{attribute 'Tc2GvlVarNames'}
{attribute 'strict'}
//Tipologia di Magazzino Falde
TYPE e_Tipo_Magazzino_Falde :
(
	NOT_DEFINED				:= -1,
	(* Magazzino Falde Per Pallettizzatore PACCHI*)
	//MAGAZZINO_FALDE_CENTRO_FISSO 		:= 1, //LA Y DI PRELIEVO RIMANE COSTANTE PER OGNI FORMATO
	//MAGAZZINO_FALDE_CENTRO_VARIABILE  	:= 2, //LA Y DI PRELIEVO SI ADATTA AL FORMATO DELLA FALDA
	
	(* Magazzino Falde per Pallettizzatore LASTRE*)
	MAGAZZINO_FALDE_IN_WA		 := 10, 	(* Identifica che il magazzino delle falde è una WorkArea *) 
	MAGAZZINO_FALDE_IN_PP		 := 20	 	(* Identifica che il magazzino delle falde è un Pick-Point, quindi elemento statico non asservito da LGV *) 

);
END_TYPE
//  NOT_DEFINED = '-1'

(* stored: Version 1.1.0.1, ProductVersion 3.1.4024.11
   EnumerationTextList e_Tipo_Magazzino_Falde: Id {26c1fc94-ade3-466c-b12e-2668dbcd11dd} *)
